FUNCTION alg_g_w_w: LREAL
{ S7_Optimized_Access := 'true' }
    VAR_INPUT
        state: STATE;
    END_VAR

BEGIN
    alg_g_w_w := state.curTime;
END_FUNCTION
